FUNCTION_BLOCK LOGGER_862393804 (* Logs a message using the logging subsystem of the runtime *)
  (* Standard: 61499-2 *)
  (* Version 1.0, 2010-11-04, medusta, nxtControl GmbH, Initial Version *)
  PACKAGE Main;
  (* Compiler Cpp *)
  {SET_ATTRIBUTE(Runtime.FBType.ImplementingType, Runtime.System#DYNGEN_LOGGER)}
  {SET_ATTRIBUTE(Configuration.GenericFBType.InterfaceParams, Runtime.System#CNT:=10)}
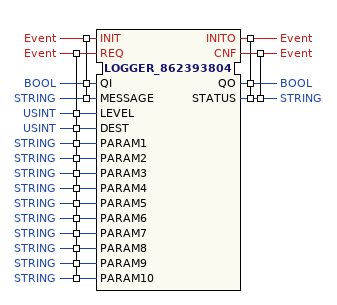
  EVENT_INPUT
    INIT WITH QI, MESSAGE; (* Initialization request *)
    REQ WITH LEVEL, PARAM1, PARAM2, PARAM3, PARAM4, PARAM5, PARAM6, PARAM7, PARAM8, PARAM9, PARAM10, DEST; (* Log request *)
  END_EVENT
  EVENT_OUTPUT
    INITO WITH QO, STATUS; (* Initialization confirmation event *)
    CNF WITH STATUS; (* Log request confirmation *)
  END_EVENT
  VAR_INPUT
    QI : BOOL; (* Input event qualifier *)
    MESSAGE : STRING; (* Logged message. ${1} inserts the value of PARAM1 etc. After this expansion the message can contain max. 256 characters. *)
    LEVEL : USINT; (* Log level *) {SET_ATTRIBUTE(ParameterEditor, ComboBox{Enums=Debug = 0|Info = 1|Warning = 2|Error = 3$})}
    DEST : USINT; (* Log destination *) {SET_ATTRIBUTE(ParameterEditor, ComboBox{Enums=Cyclic = 0|Sporadic = 1$})}
    PARAM1 : STRING; (* Parameter that can be used in the logged message. *)
    PARAM2 : STRING; (* Parameter that can be used in the logged message. *)
    PARAM3 : STRING; (* Parameter that can be used in the logged message. *)
    PARAM4 : STRING; (* Parameter that can be used in the logged message. *)
    PARAM5 : STRING; (* Parameter that can be used in the logged message. *)
    PARAM6 : STRING; (* Parameter that can be used in the logged message. *)
    PARAM7 : STRING; (* Parameter that can be used in the logged message. *)
    PARAM8 : STRING; (* Parameter that can be used in the logged message. *)
    PARAM9 : STRING; (* Parameter that can be used in the logged message. *)
    PARAM10 : STRING; (* Parameter that can be used in the logged message. *)
  END_VAR
  VAR_OUTPUT
    QO : BOOL; (* Output event qualifier *)
    STATUS : STRING; (* Status. *)
  END_VAR
  EC_STATES
    START;
  END_STATES
END_FUNCTION_BLOCK
